// TwinCAT 3 PLC project Untitled1
// ProgramVersion: 3.1.4024.0
// libraries:
//   Tc2_Standard, * (Beckhoff Automation GmbH)
//   Tc2_System, * (Beckhoff Automation GmbH)
//   Tc3_Module, * (Beckhoff Automation GmbH)
// project tree:
//   DUTs/ MyStruct.TcDUT
//   / PlcTask.TcTTO
//   POUs/ MAIN.TcPOU
// real-time tasks:
//   TASK PlcTask: cycle T#10ms, priority 20, ADS port 350

CONFIGURATION Untitled1
    RESOURCE PLC ON TwinCAT3
        TASK PlcTask(INTERVAL := T#10ms, PRIORITY := 20);
        PROGRAM MAIN WITH PlcTask : MAIN;
    END_RESOURCE
END_CONFIGURATION

// ---- DUTs/MyStruct.TcDUT
TYPE MyStruct :
STRUCT
	Par1 : INT;
	Par2 : INT;
END_STRUCT
END_TYPE

// ---- POUs/MAIN.TcPOU
PROGRAM MAIN
VAR
	TestStruct : MyStruct;
	MyRef : REFERENCE TO MyStruct;
	Test1 : INT;
	Test2 : INT;
	Test3 : INT;
	Test4 : INT;
	Run : INT;
	i : UINT;
	sIP        : STRING(255) := 'abc';
	sIP2        : STRING := 'abc';
test : UINT;	
END_VAR

IF Run = 0 THEN
	MyRef REF= TestStruct;
	TestStruct.Par1 := 1;
	TestStruct.Par2 := 2;
	Test1 := MyRef.Par1;
	MyRef.Par2 := 3;
	Test2 := MyRef.Par2;
	MyRef.Par1 := MyRef.Par2 + 1;
	Test3 := MyRef.Par1;
	Run := 1;
END_IF

IF sIP = sIP2 THEN
	i := 2;
END_IF

test := REAL_TO_UINT(67533.53);

END_PROGRAM
